Universal Robots PolyScope program: 20240924vision-J180_400-L3000_3000.urp

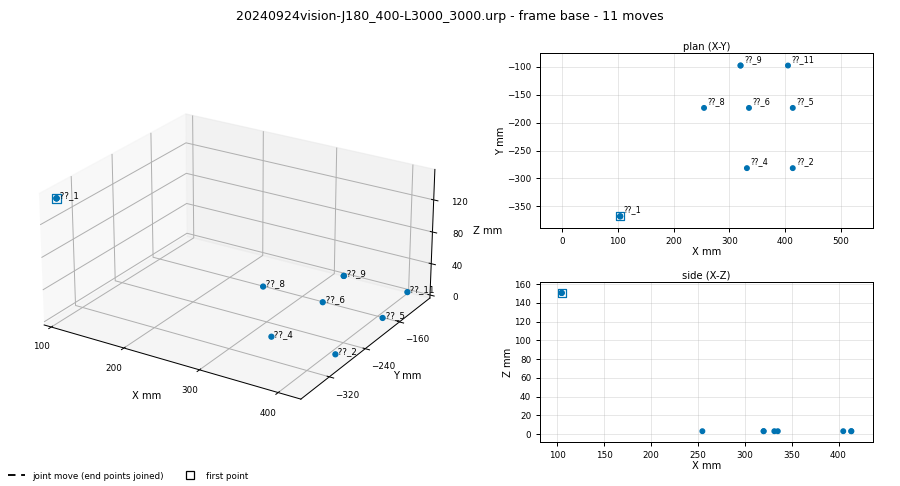
[picture p0: tool path of 20240924vision-J180_400-L3000_3000.urp in frame base, 11 of 32 moves have a stored position in this frame; points joined in program order, loops and branches not executed]
Program 20240924vision-J180_400-L3000_3000 (installation=20240827 directory=/programs/Demos/vision createdIn=5.13.1 lastSavedIn=5.15.1 robotSerialNumber=20245500285)
Calibrated DH parameters: a=[0.000097, -0.210459, -0.026602, 0.000137, 0.000078, 0]; d=[0.162601, 254.180657, -54.076236, -199.970743, 0.099615, 0.099684]; alpha=[1.569796, -0.001455, 0.001957, 1.570525, -1.571561, 0]; deltaTheta=[0, -1.053331, 8.839472, -1.50296, 0.000002, 0]
InitVariablesNode
Robot Program (runOnlyOnce=false)
  MoveJ speed 180 deg/s, acceleration 400 deg/s^2 (useActiveTCP=true positionType=JointAngles) feature=Base
    Waypoint 路点_1: TCP in base x=104.511 y=-367.887 z=150.56 mm, rx=-1.9493 ry=-1.8262 rz=-0.6048 rad; joints [85.471, -80.224, 100.082, -75.625, -90.165, 89.439] deg; TCP offset x=-0.17 y=0 z=192.95 mm, rx=0 ry=0 rz=0 rad
  Script: vision = rpc_factory("xmlrpc","http://192.168.1.7:9121/RPC2")
  Script: gripper = rpc_factory("xmlrpc","http://192.168.1.7:9120/RPC2")
  Script: gripper.open()
  SuppressedNode
    Wait Sleep waitTime=1
  SuppressedNode
    Script: usb.adaptiveClose()
  SuppressedNode
    Halt
  n := 1
  Loop Forever
    MoveJ speed 180 deg/s, acceleration 400 deg/s^2 (useActiveTCP=true) feature=Base
      Waypoint 路点_1: TCP in base x=104.511 y=-367.887 z=150.56 mm, rx=-1.9493 ry=-1.8262 rz=-0.6048 rad; joints [85.471, -80.224, 100.082, -75.625, -90.165, 89.439] deg
    Popup Message (haltProgram=false message=photo inputType=Text)
    trszzz := 0.06
    campose := get_actual_tcp_pose()
    'USB'
    Script: vision.take_photo(campose)
    'USB'
    articlenum := vision.get_obj_num()
    Popup Message (haltProgram=false message=123 inputType=Text)
    Loop While (checkContinuously=false) expression=n≤articlenum
      SuppressedNode
        obj_num :=  (valueSource=Operator valueType=Integer)
      obj_num := n
      SuppressedNode
        Popup Message (haltProgram=false message=12 inputType=Text)
      pose := p[0.0,0.0,0.0,2.221,2.221,0.004]
      SuppressedNode
        Script: var_2 = move.move_pose(obj_num)
      var_2 := vision.get_obj_pose(obj_num)
      SuppressedNode
        Script: var_2 = move.move_pose(n)
      Script: pose[0]=var_2[0]
      Script: pose[1]=var_2[1]
      Script: pose[2]=var_2[2]
      Popup Message (haltProgram=false inputType=Variable) variable(name=pose)
      MoveL speed 3000 mm/s, acceleration 3000 mm/s^2 (useActiveTCP=true) feature=Base
        Waypoint Variable (Variable): variable(name=pose)
      Script: pose[2]=var_2[2] - 0.035
      If pose[2] ≥ 0.003
        MoveL speed 3000 mm/s, acceleration 3000 mm/s^2 (useActiveTCP=true) feature=Base
          Waypoint Variable (Variable): variable=pose
          Script: gripper.adaptiveClose()
      ElseIf pose[2] < 0.003
        Script: pose[2] = 0.003
        MoveL speed 3000 mm/s, acceleration 3000 mm/s^2 (useActiveTCP=true) feature=Base
          Waypoint Variable (Variable): variable=pose
          Script: gripper.adaptiveClose()
      SuppressedNode
        Else 
          Popup Warning (haltProgram=false message=pose_z too low inputType=Text)
      Popup Message (haltProgram=false inputType=Variable) variable=pose
      h1 := pose
      SuppressedNode
        MoveL speed 3000 mm/s, acceleration 1000 mm/s^2 (useActiveTCP=true) feature=Base
          Waypoint Variable (Variable): variable=pose
      SuppressedNode
        Script: gripper.adaptiveClose()
      Script: pose[2]=var_2[2] + trszzz
      SuppressedNode
        Script: pose[2]=var_2[2] + 0.1
      MoveL speed 3000 mm/s, acceleration 3000 mm/s^2 (useActiveTCP=true) feature=Base
        Waypoint Variable (Variable): variable=pose
      SuppressedNode
        MoveJ speed 150 deg/s, acceleration 100 deg/s^2 (useActiveTCP=true) feature=Base
          Waypoint 路点_3: TCP in base x=148.551 y=-281.526 z=149.247 mm, rx=2.2211 ry=2.2211 rz=0.0029 rad; joints [92.81, -116.498, 131.46, -104.954, -89.899, 92.941] deg
          SuppressedNode
            trs1 := pose_add(路点_4, p[0,0,0.2,0,0,0])
      trs1 := pose_add(路点_4, p[0,0,trszzz,0,0,0])
      SuppressedNode
        trs1 := pose_add(路点_4, p[0,0,0.2,0,0,0])
      tar1 := pose_add(路点_4, p[0,0,h1[2],0,0,0])
      Popup Message (haltProgram=false inputType=Variable) variable(name=tar1)
      tar1 := 路点_4
      Script: tar1[2]=h1[2]
      If n == 1
        MoveL speed 3000 mm/s, acceleration 3000 mm/s^2 (useActiveTCP=true) feature=Base
          Waypoint Variable (Variable): variable(name=trs1)
        MoveL speed 3000 mm/s, acceleration 3000 mm/s^2 (useActiveTCP=true) feature=Base
          Popup Message (haltProgram=false message=1111111111 inputType=Text)
          Waypoint Variable (Variable): variable(name=tar1)
          Popup Message (haltProgram=false message=1111111111 inputType=Text)
          If 0
            Waypoint 路点_4 referenceName=路点_4: TCP in base x=331.461 y=-281.525 z=3 mm, rx=2.2211 ry=2.2211 rz=0.0029 rad; joints [121.608, -83.342, 130.91, -137.615, -89.956, 121.753] deg
          Popup Message (haltProgram=false message=000000 inputType=Text)
          SuppressedNode
            Waypoint 路点_4: TCP in base x=331.461 y=-281.525 z=3 mm, rx=2.2211 ry=2.2211 rz=0.0029 rad; joints [121.608, -83.342, 130.91, -137.615, -89.956, 121.753] deg
          Script: gripper.open()
        MoveL speed 3000 mm/s, acceleration 3000 mm/s^2 (useActiveTCP=true) feature=Base
          Waypoint Variable (Variable): variable=trs1
      trs2 := pose_add(路点_2, p[0,0,trszzz,0,0,0])
      SuppressedNode
        trs2 := pose_add(路点_2, p[0,0,0.2,0,0,0])
      If n == 2
        MoveL speed 3000 mm/s, acceleration 3000 mm/s^2 (useActiveTCP=true) feature=Base
          Waypoint Variable (Variable): variable(name=trs2)
        MoveL speed 3000 mm/s, acceleration 3000 mm/s^2 (useActiveTCP=true) feature=Base
          Waypoint 路点_2 referenceName=路点_2: TCP in base x=413.578 y=-281.55 z=3 mm, rx=2.2212 ry=2.221 rz=0.0029 rad; joints [130.122, -75.511, 120.827, -135.378, -89.965, 130.285] deg
          Script: gripper.open()
        MoveL speed 3000 mm/s, acceleration 3000 mm/s^2 (useActiveTCP=true) feature=Base
          Waypoint Variable (Variable): variable=trs2
      trs3 := pose_add(路点_5, p[0,0,trszzz,0,0,0])
      SuppressedNode
        trs3 := pose_add(路点_5, p[0,0,0.2,0,0,0])
      If n == 3
        MoveL speed 3000 mm/s, acceleration 3000 mm/s^2 (useActiveTCP=true) feature=Base
          Waypoint Variable (Variable): variable(name=trs3)
        MoveL speed 3000 mm/s, acceleration 3000 mm/s^2 (useActiveTCP=true) feature=Base
          Waypoint 路点_5 referenceName=路点_5: TCP in base x=413.621 y=-173.641 z=3 mm, rx=2.221 ry=2.2212 rz=0.0029 rad; joints [139.755, -81.637, 128.862, -137.305, -89.965, 139.9] deg
          Script: gripper.open()
        MoveL speed 3000 mm/s, acceleration 3000 mm/s^2 (useActiveTCP=true) feature=Base
          Waypoint Variable (Variable): variable=trs3
      trs4 := pose_add(路点_6, p[0,0,trszzz,0,0,0])
      SuppressedNode
        trs4 := pose_add(路点_6, p[0,0,0.2,0,0,0])
      If n == 4
        MoveL speed 3000 mm/s, acceleration 3000 mm/s^2 (useActiveTCP=true) feature=Base
          Waypoint Variable (Variable): variable(name=trs4)
        MoveL speed 3000 mm/s, acceleration 3000 mm/s^2 (useActiveTCP=true) feature=Base
          Waypoint 路点_6 referenceName=路点_6: TCP in base x=335.16 y=-173.643 z=3 mm, rx=2.2211 ry=2.2211 rz=0.0029 rad; joints [131.722, -91.143, 139.321, -138.241, -89.956, 131.857] deg
          Script: gripper.open()
        MoveL speed 3000 mm/s, acceleration 3000 mm/s^2 (useActiveTCP=true) feature=Base
          Waypoint Variable (Variable): variable=trs4
      trs5 := pose_add(路点_8, p[0,0,trszzz,0,0,0])
      SuppressedNode
        trs5 := pose_add(路点_8, p[0,0,0.2,0,0,0])
      If n == 5
        MoveL speed 3000 mm/s, acceleration 3000 mm/s^2 (useActiveTCP=true) feature=Base
          Waypoint Variable (Variable): variable(name=trs5)
        MoveL speed 3000 mm/s, acceleration 3000 mm/s^2 (useActiveTCP=true) feature=Base
          Waypoint 路点_8 referenceName=路点_8: TCP in base x=254.659 y=-173.63 z=3 mm, rx=2.2212 ry=2.2211 rz=0.0029 rad; joints [119.834, -102.953, 148.816, -135.903, -89.943, 119.958] deg
          Script: gripper.open()
        MoveL speed 3000 mm/s, acceleration 3000 mm/s^2 (useActiveTCP=true) feature=Base
          Waypoint Variable (Variable): variable=trs5
      trs6 := pose_add(路点_9, p[0,0,trszzz,0,0,0])
      SuppressedNode
        trs6 := pose_add(路点_9, p[0,0,0.2,0,0,0])
      If n == 6
        MoveL speed 3000 mm/s, acceleration 3000 mm/s^2 (useActiveTCP=true) feature=Base
          Waypoint Variable (Variable): variable(name=trs6)
        MoveL speed 3000 mm/s, acceleration 3000 mm/s^2 (useActiveTCP=true) feature=Base
          Waypoint 路点_9 referenceName=路点_9: TCP in base x=320.033 y=-97.716 z=3 mm, rx=2.2212 ry=2.2212 rz=0.0029 rad; joints [139.32, -98.009, 145.306, -137.371, -89.952, 139.448] deg
          Script: gripper.open()
        MoveL speed 3000 mm/s, acceleration 3000 mm/s^2 (useActiveTCP=true) feature=Base
          Waypoint Variable (Variable): variable=trs6
      trs7 := pose_add(路点_9, p[0,0,trszzz,0,0,0])
      SuppressedNode
        trs7 := pose_add(路点_9, p[0,0,0.2,0,0,0])
      If n == 7
        MoveL speed 3000 mm/s, acceleration 3000 mm/s^2 (useActiveTCP=true) feature=Base
          Waypoint Variable (Variable): variable(name=trs7)
        MoveL speed 3000 mm/s, acceleration 3000 mm/s^2 (useActiveTCP=true) feature=Base
          Waypoint 路点_9 referenceName=路点_9: TCP in base x=320.033 y=-97.716 z=3 mm, rx=2.2212 ry=2.2212 rz=0.0029 rad; joints [139.32, -98.009, 145.306, -137.371, -89.952, 139.448] deg
          Script: gripper.open()
        MoveL speed 3000 mm/s, acceleration 3000 mm/s^2 (useActiveTCP=true) feature=Base
          Waypoint Variable (Variable): variable=trs7
      trs8 := pose_add(路点_11, p[0,0,trszzz,0,0,0])
      SuppressedNode
        trs8 := pose_add(路点_11, p[0,0,0.2,0,0,0])
      If n == 8
        MoveL speed 3000 mm/s, acceleration 3000 mm/s^2 (useActiveTCP=true) feature=Base
          Waypoint Variable (Variable): variable(name=trs8)
        MoveL speed 3000 mm/s, acceleration 3000 mm/s^2 (useActiveTCP=true) feature=Base
          Waypoint 路点_11 referenceName=路点_11: TCP in base x=405.013 y=-97.732 z=3 mm, rx=2.2212 ry=2.2211 rz=0.0029 rad; joints [147.586, -85.701, 133.648, -138.037, -89.967, 147.73] deg
          Script: gripper.open()
        MoveL speed 3000 mm/s, acceleration 3000 mm/s^2 (useActiveTCP=true) feature=Base
          Waypoint Variable (Variable): variable=trs8
      trs9 := pose_add(路点_11, p[0,0,trszzz,0,0,0])
      SuppressedNode
        trs9 := pose_add(路点_11, p[0,0,0.2,0,0,0])
      SuppressedNode
        If n == 9
          MoveL speed 3000 mm/s, acceleration 1000 mm/s^2 (useActiveTCP=true) feature=Base
            Waypoint Variable (Variable): variable(name=trs9)
          MoveL speed 3000 mm/s, acceleration 1000 mm/s^2 (useActiveTCP=true) feature=Base
            Waypoint 路点_11 referenceName=路点_11: TCP in base x=405.013 y=-97.732 z=3 mm, rx=2.2212 ry=2.2211 rz=0.0029 rad; joints [147.586, -85.701, 133.648, -138.037, -89.967, 147.73] deg
            Script: gripper.open()
          MoveL speed 3000 mm/s, acceleration 1000 mm/s^2 (useActiveTCP=true) feature=Base
            Waypoint Variable (Variable): variable=trs9
      n := n + 1
    MoveJ speed 180 deg/s, acceleration 400 deg/s^2 (useActiveTCP=true) feature=Base
      Waypoint 路点_1: TCP in base x=104.511 y=-367.887 z=150.56 mm, rx=-1.9493 ry=-1.8262 rz=-0.6048 rad; joints [85.471, -80.224, 100.082, -75.625, -90.165, 89.439] deg; TCP offset x=-0.17 y=0 z=192.95 mm, rx=0 ry=0 rz=0 rad
      n := 1
